FUNCTION_BLOCK XtsTmsSwitch IMPLEMENTS ITF_TmsSwitch
VAR_INPUT
	StateMachine : IPmlStateMachine;
END_VAR
VAR_OUTPUT
END_VAR
VAR
	positionState : SwitchState := SwitchState.Middle;
	UpPosition : MC_LREAL := 100.0;
	MiddlePosition : MC_LREAL := 200.0;
	DownPosition : MC_LREAL := 300.0;
	SwitchVelocity : MC_LREAL := 100.0;
	switchAxis : MC2_Axis_Base;	
	State :(
        Init,                                               
		Ready,                                 
        Enabling,
		Enabled,
		Resetting,
		Running,
		Disabling); 
END_VAR

CASE State OF
	Init:
		IF NOT switchAxis.hasError() THEN
			State := Ready;
		END_IF
		
	Ready:
		IF StateMachine.GetCurrentState() = E_PMLState.ePMLState_Clearing THEN
			IF switchAxis.EnableAxis() THEN
				State := Enabling;
			END_IF
		END_IF	
		
	Enabling:
		IF switchAxis.isEnabled() THEN
			State := Enabled;
		END_IF
		
	Enabled:
		IF StateMachine.GetCurrentState() = E_PMLState.ePMLState_Resetting THEN
			IF switchAxis.MoveTo(Position := MiddlePosition, Velocity := 100.0) THEN
				State := Resetting;
			END_IF
		END_IF
		
	Resetting:
		IF switchAxis.isAtPosition(position := MiddlePosition) THEN
			State := Running;
		END_IF	
	
	Running:	
		
	Disabling:

END_CASE

switchAxis();

METHOD PUBLIC MoveTo : BOOL
VAR_INPUT
	positionState : SwitchState;
END_VAR
CASE positionState OF
	SwitchState.Down:
		IF NOT isAtPosition(position := DownPosition) THEN
			IF NOT axesMoveTo.Busy THEN
				axesMoveTo.MoveTo(Position := DownPosition, Velocity := SwitchVelocity);
				MoveTo := TRUE;
			END_IF
		END_IF
	SwitchState.Middle:
		IF NOT isAtPosition(position := MiddlePosition) THEN
			IF NOT axesMoveTo.Busy THEN
				axesMoveTo.MoveTo(Position := MiddlePosition, Velocity := SwitchVelocity);
				MoveTo := TRUE;
			END_IF
		END_IF
	SwitchState.Up:
		IF NOT isAtPosition(position := UpPosition) THEN
			IF NOT axesMoveTo.Busy THEN
				axesMoveTo.MoveTo(Position := UpPosition, Velocity := SwitchVelocity);
				MoveTo := TRUE;
			END_IF
		END_IF
END_CASE
END_METHOD

PROPERTY PUBLIC Switch : SwitchState
GET
Switch := positionState;
END_GET
END_PROPERTY

END_FUNCTION_BLOCK

(* stored: Version 1.1.0.1, ProductVersion 3.1.4024.11
   POU XtsTmsSwitch: Id {73ef316f-86b5-4cc1-962a-15251e072db1}, SpecialFunc None
   Method MoveTo: Id {fd17c823-afe7-4820-9dad-912e69242e2b}
   Property Switch: Id {cea7677b-4e3e-436d-9a14-24ba96282e4e}
   Get Get: Id {955c8029-4c60-4733-8b6b-b2d2d74760a8} *)
